# EPICS StreamDevice protocol: IC101App/src/IC101.proto
########################################################################
# StreamDevice protocol for the IC101.                                 #
########################################################################

InTerminator = CR LF;
OutTerminator = LF;
replytimeout = 500;
readtimeout  = 1000;
locktimeout = 60000;

# Set/Query Maximum *External* High Voltage in Volts
setHVMax {
	InTerminator = LF ACK;
	out "CONFigure:HIVOltage:MAXvalue %d";
	in "CONFigure:HIVOltage:MAXvalue %d";
}

getHVMax {
	out "CONFigure:HIVOltage:MAXvalue?";
	in "CONFigure:HIVOltage:MAXvalue?", LF ACK, "%d";
}

# Set/Query External High Voltage in Volts
setHV {
	InTerminator = LF ACK;
	out "CONFigure:HIVOltage:SET %d";
	in "CONFigure:HIVOltage:SET %d";
}

getHV {
	out "CONFigure:HIVOltage:SET?";
	in "CONFigure:HIVOltage:SET?", LF ACK, "%d";
}

# check for ext voltage - Bell returns 0 and ACK returns 1
checkHV {
	out "CONFigure:HIVOltage:SET?";
	in "CONFigure:HIVOltage:SET?\n%{\7|\6}";
	ExtraInput = IGNORE;
}

# Query the last measured current data in amps.
readCurrents {
	replytimeout = 100;
	readtimeout  = 65001;  #echos command and waits for values
	locktimeout = 65005;
	InTerminator = CR LF;
	out "READ:CURRent?";
 	##I100 $1=Dev $2=time $3=OVR
 	in "READ:CURRent?\n\x06%(\$1:\$2.VAL)e %(\$1:\$2.EGU)c,%e %(EGU)c,%(\$1:\$3.VAL)i";
}

# Set/Query current Range
setRange {
	InTerminator = LF ACK;
	out "CONFigure:RANGe %e";
	in "CONFigure:RANGe %e";
}

getRange {
	out "CONFigure:RANGe?";
	in "CONFigure:RANGe?\n\x06%e %(EGU)c";
	@readtimeout {
		IN "CONFigure:RANGe?",LF BEL;
	}
}

# Set/Query current Range
setPeriod {
	InTerminator = LF ACK;
	out "CONFigure:PERiod %e";
	in "CONFigure:PERiod %e";
}

getPeriod {
	out "CONFigure:PERiod?";
	in "CONFigure:PERiod?\n\x06%e %(EGU)c";
}

#EOF
